SUBAPPLICATION Uebung_204b_AX (* Interlock: ILOCK_CONFLICT_TRIP_AX (Motor-Sicherheitsabschaltung via Adapter) *)
  (* Standard: 61499-2; Description: Copyright (c) 2023 Meisterschulen am Ostbahnhof This program and the accompanying materials are made available under the terms of the Eclipse Public License 2.0 which is available at https://www.eclipse.org/legal/epl-2.0/ SPDX-License-Identifier: EPL-2.0 *)
  (* Version 1.0, 2026-04-19, Franz Höpfinger, Meisterschulen am Ostbahnhof, initial API and implementation and/or initial documentation *)
  PACKAGE Uebungen;
  IMPORT logiBUS::io::DI::logiBUS_DI::Input_I1;
  IMPORT logiBUS::io::DI::logiBUS_DI::Input_I2;
  IMPORT logiBUS::io::DI::logiBUS_DI::Input_I3;
  IMPORT logiBUS::io::DI::logiBUS_DI_Events::BUTTON_SINGLE_CLICK;
  IMPORT logiBUS::io::DQ::logiBUS_DO::Output_Q4;
  IMPORT logiBUS::io::DQ::logiBUS_DO::Output_Q5;
  IMPORT logiBUS::io::DQ::logiBUS_DO::Output_Q56;
  IMPORT logiBUS::io::DQ::logiBUS_DO::Output_Q6;
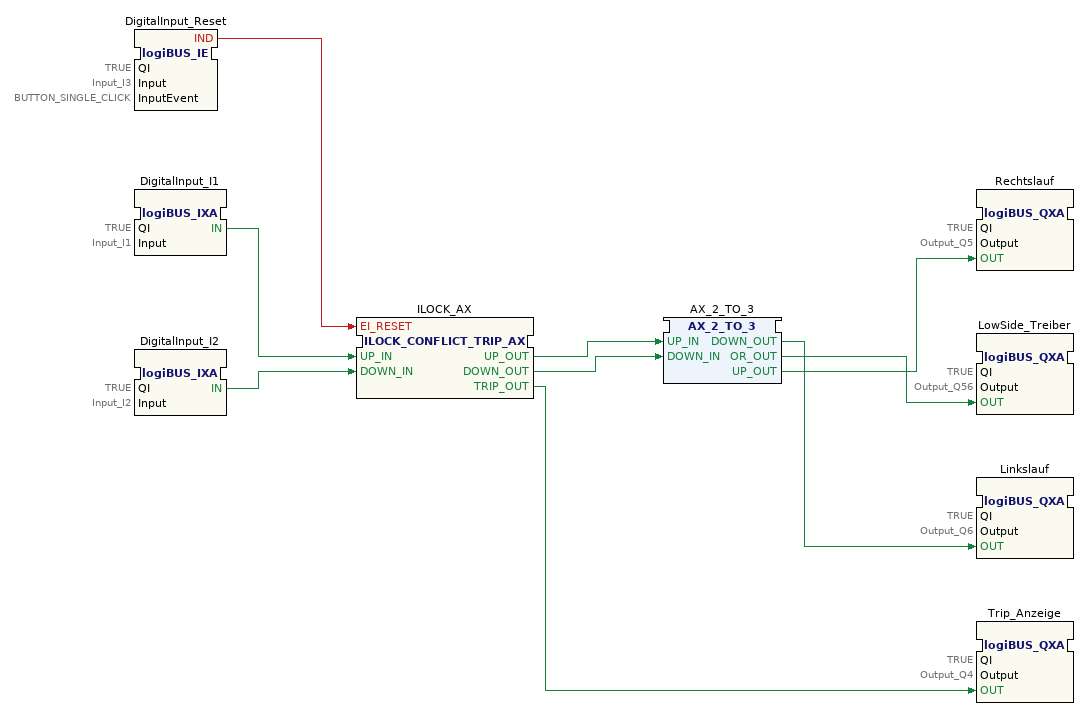
  FBS
    DigitalInput_I1 : logiBUS::io::DI::logiBUS_IXA(QI := TRUE, Input := Input_I1);
    DigitalInput_I2 : logiBUS::io::DI::logiBUS_IXA(QI := TRUE, Input := Input_I2);
    ILOCK_AX : logiBUS::signalprocessing::interlock::ILOCK_CONFLICT_TRIP_AX;
    Rechtslauf : logiBUS::io::DQ::logiBUS_QXA(QI := TRUE, Output := Output_Q5);
    Linkslauf : logiBUS::io::DQ::logiBUS_QXA(QI := TRUE, Output := Output_Q6);
    Trip_Anzeige : logiBUS::io::DQ::logiBUS_QXA(QI := TRUE, Output := Output_Q4);
    LowSide_Treiber : logiBUS::io::DQ::logiBUS_QXA(QI := TRUE, Output := Output_Q56);
    DigitalInput_Reset : logiBUS::io::DI::logiBUS_IE(QI := TRUE, Input := Input_I3, InputEvent := BUTTON_SINGLE_CLICK);
  END_FBS
  SUBAPPS
    AX_2_TO_3 : MyLib::sys::AX_2_TO_3;
  END_SUBAPPS
  EVENT_CONNECTIONS
    DigitalInput_Reset.IND TO ILOCK_AX.EI_RESET;
  END_CONNECTIONS
  ADAPTER_CONNECTIONS
    DigitalInput_I1.IN TO ILOCK_AX.UP_IN;
    DigitalInput_I2.IN TO ILOCK_AX.DOWN_IN;
    ILOCK_AX.UP_OUT TO AX_2_TO_3.UP_IN;
    ILOCK_AX.DOWN_OUT TO AX_2_TO_3.DOWN_IN;
    ILOCK_AX.TRIP_OUT TO Trip_Anzeige.OUT;
    AX_2_TO_3.DOWN_OUT TO Linkslauf.OUT;
    AX_2_TO_3.OR_OUT TO LowSide_Treiber.OUT;
    AX_2_TO_3.UP_OUT TO Rechtslauf.OUT;
  END_CONNECTIONS
END_SUBAPPLICATION
